// TIA Portal V16 export
// export: Created 2024-09-05T17:36:33.8494984Z, ExportSetting WithDefaults, DisplayName Totally Integrated Automation Portal, DisplayVersion V16 Update 6, DisplayName TIA Portal Version Control Interface, DisplayVersion V16 Update 2, DisplayName TIA Portal Openness, DisplayVersion V16 Update 6, DisplayName STEP 7 Professional, DisplayVersion V16 Update 6, DisplayName STEP 7 Safety, DisplayVersion V16, DisplayName WinCC Advanced, DisplayVersion V16 Update 6
VAR_GLOBAL   // PLC tag table "st3 - jig"
   i3partPresent AT %I27.5 : Bool;   // jig
   qRiveting1Start AT %Q11.1 : Bool;   // ST3 - Baltec: Start riveting
   qRiveting1Bit0 AT %Q11.2 : Bool;   // ST3 - Baltec: Program number BCD 1
   qRiveting1Bit1 AT %Q11.3 : Bool;   // ST3 - Baltec: Program number BCD 2
   qRiveting1Bit2 AT %Q11.4 : Bool;   // ST3 - Baltec: Program number BCD 4
   qRiveting1Bit3 AT %Q11.5 : Bool;   // ST3 - Baltec: Program number BCD 8
   qRiveting1Bit4 AT %Q11.6 : Bool;   // ST3 - Baltec: Program number BCD 16
   qRiveting2Start AT %Q12.1 : Bool;   // ST3 - Baltec: Start riveting
   qRiveting2Bit0 AT %Q12.2 : Bool;   // ST3 - Baltec: Program number BCD 1
   qRiveting2Bit1 AT %Q12.3 : Bool;   // ST3 - Baltec: Program number BCD 2
   qRiveting2Bit2 AT %Q12.4 : Bool;   // ST3 - Baltec: Program number BCD 4
   qRiveting2Bit3 AT %Q12.5 : Bool;   // ST3 - Baltec: Program number BCD 8
   qRiveting2Bit4 AT %Q12.6 : Bool;   // ST3 - Baltec: Program number BCD 16
   iRivetingReady1 AT %I12.0 : Bool;
   iRivetingH1ok1 AT %I12.1 : Bool;
   iRivetingH2ok1 AT %I12.2 : Bool;
   iRivetingTimeOk1 AT %I12.3 : Bool;
   iRivetingZ1ok1 AT %I12.4 : Bool;
   iRivetingNoError1 AT %I12.5 : Bool;
   iRivetingReady2 AT %I13.0 : Bool;
   iRivetingH1ok2 AT %I13.1 : Bool;
   iRivetingH2ok2 AT %I13.2 : Bool;
   iRivetingTimeOk2 AT %I13.3 : Bool;
   iRivetingZ1ok2 AT %I13.4 : Bool;
   iRivetingNoError2 AT %I13.5 : Bool;
   qFriedrich1_setup_mode AT %Q0.3 : Bool;
   qFriedrich2_setup_mode AT %Q0.4 : Bool;
END_VAR
